{attribute addProperty BoxType "EK1100-0000-0018"}
{attribute addProperty Id "Beckhoff_ER1xxxEK1122Beckhoff_ER1xxxEK1122_B47283563856482"}
{attribute addProperty CRC "6094411"}
{attribute addProperty SizeInBites "3856"}
{attribute addProperty SizeInBytes "482"}
TYPE Beckhoff_ER1xxx_005CFE4B EXTENDS EK1100_179A0949 :
STRUCT
	{attribute addProperty Name "Beckhoff_ER1xxxEK1122"}
	Beckhoff_ER1xxxEK1122 : Beckhoff_ER1xxxEK1122_B4728356;
END_STRUCT
END_TYPE

(* stored: Version 1.2.0.0, ProductVersion 3.1.4024.9
   DUT Beckhoff_ER1xxx_005CFE4B: Id {4e9d66dd-8e63-4148-81bd-67e92fc000d2} *)
